// TIA Portal V17 export
// export: Created 2025-05-22T06:01:20.0490676Z, ExportSetting WithDefaults, DisplayName Totally Integrated Automation Portal, DisplayVersion V17 Update 8, DisplayName TIA Portal Openness, DisplayVersion V17 Update 8, DisplayName TIA Portal Version Control Interface, DisplayVersion V17, DisplayName SINAMICS Startdrive Advanced, DisplayVersion V17 SP2, DisplayName SINAMICS Startdrive G110M, G120, G120C, G120D, G120P, G115D, DisplayVersion V17 SP2, DisplayName SINAMICS Startdrive G130, G150, S120, S150, SINAMICS MV, S210, DisplayVersion V17 SP2, DisplayName STEP 7 Professional, DisplayVersion V17 Update 8, DisplayName SINUMERIK ONE STEP 7 Toolbox, DisplayVersion V17 Update 12, DisplayName SINUMERIK ONE PLC Basic Program Plus, DisplayVersion V17 Update 12, DisplayName SINUMERIK 840D sl STEP 7 Toolbox, DisplayVersion V17 Update 12, DisplayName STEP 7 Safety, DisplayVersion V17 Update 6, DisplayName WinCC Advanced, DisplayVersion V17 Update 8
DATA_BLOCK "DB10404_U2_STA_3_PRESSURE_SENSOR"   // DB10404
{ DB_Accessible_From_OPC_UA := 'FALSE' }
VERSION : 0.1
// stored: AutoNumber false, DBAccessibleFromOPCUA false, DBAccessibleFromWebserver true, InstanceOfName FB10400_PRESSURE_SENSOR, InstanceOfType FB
"FB10400_PRESSURE_SENSOR"
   // VAR_INPUT
   //    SENSOR_VALUE_I : Int;
   //    STATION_CYCLE_RUNNING : Bool;
   // END_VAR
   // VAR_OUTPUT
   //    LOW_PRESSURE_ALARM : Bool;
   //    HIGH_PRESSURE_ALARM : Bool;
   //    LOW_PRESSURE_WARNING : Bool;
   //    HIGH_PRESSURE_WARNING : Bool;
   // END_VAR
   // VAR RETAIN
   //    HMI : Struct
   //       HIGH_LIMIT_ALARM_VALUE : Real := 1000.0;
   //       HIGH_LIMIT_WARNING_VALUE : Real := 1000.0;
   //       LOW_LIMIT_ALARM_VALUE : Real := -1000.0;
   //       LOW_LIMIT_WARNING_VALUE : Real := -1000.0;
   //    END_STRUCT;
   //    SETTINGS : Struct
   //       NORM_MIN_VAL : Int := 0;
   //       NORM_MAX_VAL : Int := 32240;
   //       SCALE_MIN_VAL : Real := -1000.0;
   //       SCALE_MAX_VAL : Real := 1000.0;
   //       MUL_VAL : Real := 1.0;
   //       DIV_VAL : Real := 1.0;
   //       UNIT_NO : Int := 1;
   //    END_STRUCT;
   //    OUTPUT : Struct
   //       PRESSURE_VALUE : Real;
   //    END_STRUCT;
   //    INTERNAL : Struct
   //       NORMALIZED_VALUE : Real;
   //       SCALED_VALUE : Real;
   //       MULTIPLIED_VALUE : Real;
   //    END_STRUCT;
   //    ALARMS : Struct
   //       LOW_PRESSURE_ALARM : Bool;
   //       HIGH_PRESSURE_ALARM : Bool;
   //       LOW_PRESSURE_WARNING : Bool;
   //       HIGH_PRESSURE_WARNING : Bool;
   //    END_STRUCT;
   //    TIMERS : Struct
   //       ASPIRATION_LOW_ALARM_TIMER : TON_TIME;
   //       ASPIRATION_LOW_WARNING_TIMER : TON_TIME;
   //       ASPIRATION_HIGH_ALARM_TIMER : TON_TIME;
   //       ASPIRATION_HIGH_WARNING_TIMER : TON_TIME;
   //    END_STRUCT;
   // END_VAR
BEGIN
   TIMERS.ASPIRATION_LOW_ALARM_TIMER.PT := T#3s;
   TIMERS.ASPIRATION_LOW_WARNING_TIMER.PT := T#3s;
   TIMERS.ASPIRATION_HIGH_ALARM_TIMER.PT := T#3s;
   TIMERS.ASPIRATION_HIGH_WARNING_TIMER.PT := T#3s;
END_DATA_BLOCK
